// ---- VISUs/Modes/ProductionMode/V_ProductionBorgoFlaps.TcVIS
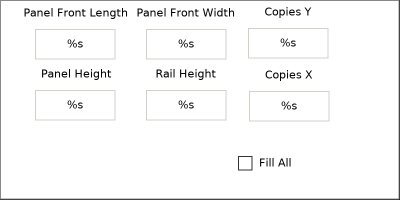
VISUALIZATION V_ProductionBorgoFlaps  // 400x200
VAR_IN_OUT
	HMI : ST_PackMLBaseModule_HMI;
	HMI_GantryXYZ : ST_GantryXYZ_HMI;
	HMI_Recipe : ST_RecipeBuilder_HMI;
END_VAR
    RoundedRectangle (0,0 400x200)
    Textfield (35,29 80x30), "%s", text variable: HMI_Recipe.Config.PanelFrontLength
        OnMouseClick: write the text variable via VisuDialogs.Numpad, min HMI_Recipe.Limits.PanelFrontLength.MinVal, max HMI_Recipe.Limits.PanelFrontLength.MaxVal
    Label (18,3 116x20), "Panel Front Length"
    Textfield (146,29 80x30), "%s", text variable: HMI_Recipe.Config.PanelFrontWidth
        OnMouseClick: write the text variable via VisuDialogs.Numpad, min HMI_Recipe.Limits.PanelFrontWidth.MinVal, max HMI_Recipe.Limits.PanelFrontWidth.MaxVal
    Label (97,3 178x20), "Panel Front Width"
    Textfield (35,90 80x30), "%s", text variable: HMI_Recipe.Config.PanelHeight
        OnMouseClick: write the text variable via VisuDialogs.Numpad, min HMI_Recipe.Limits.PanelHeight.MinVal, max HMI_Recipe.Limits.PanelHeight.MaxVal
    Label (19,64 115x20), "Panel Height"
    Textfield (146,90 80x30), "%s", text variable: HMI_Recipe.Config.RailHeightCorrection
        OnMouseClick: write the text variable via VisuDialogs.Numpad, min HMI_Recipe.Limits.RailHeightCorrection.MinVal, max HMI_Recipe.Limits.RailHeightCorrection.MaxVal
    Label (135,64 102x20), "Rail Height"
    Checkbox (236,148 72x30), "Fill All", variable: HMI_Recipe.Config.FillAll
    Textfield (249,91 80x30), "%s", text variable: HMI_Recipe.Config.RequestedCopiesX, input disabled if: MAIN.Seedra.RecipeConfig_HMI.Config.FillAll
        OnMouseClick: write the text variable via VisuDialogs.Numpad, min 1, max MAIN.Seedra.RecipeConfig_HMI.Limits.RequestedCopiesX.MaxVal
    Label (238,65 102x20), "Copies X"
    Textfield (248,28 80x30), "%s", text variable: HMI_Recipe.Config.RequestedCopiesY, input disabled if: MAIN.Seedra.RecipeConfig_HMI.Config.FillAll
        OnMouseClick: write the text variable via VisuDialogs.Numpad, min 1, max MAIN.Seedra.RecipeConfig_HMI.Limits.RequestedCopiesY.MaxVal
    Label (237,2 102x20), "Copies Y"
END_VISUALIZATION

// ---- VISUs/Modes/ProductionMode/V_ProductionBorgoWings.TcVIS
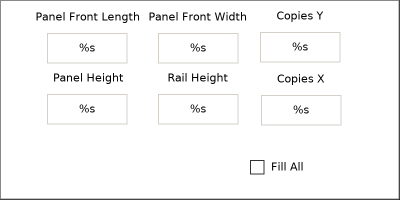
VISUALIZATION V_ProductionBorgoWings  // 400x200
VAR_IN_OUT
	HMI : ST_PackMLBaseModule_HMI;
	HMI_GantryXYZ : ST_GantryXYZ_HMI;
	HMI_Recipe : ST_RecipeBuilder_HMI;
END_VAR
    RoundedRectangle (0,0 400x200)
    Textfield (47,33 80x30), "%s", text variable: HMI_Recipe.Config.PanelFrontLength
        OnMouseClick: write the text variable via VisuDialogs.Numpad, min HMI_Recipe.Limits.PanelFrontLength.MinVal, max HMI_Recipe.Limits.PanelFrontLength.MaxVal
    Label (30,7 116x20), "Panel Front Length"
    Textfield (158,33 80x30), "%s", text variable: HMI_Recipe.Config.PanelFrontWidth
        OnMouseClick: write the text variable via VisuDialogs.Numpad, min HMI_Recipe.Limits.PanelFrontWidth.MinVal, max HMI_Recipe.Limits.PanelFrontWidth.MaxVal
    Label (109,7 178x20), "Panel Front Width"
    Textfield (47,94 80x30), "%s", text variable: HMI_Recipe.Config.PanelHeight
        OnMouseClick: write the text variable via VisuDialogs.Numpad, min HMI_Recipe.Limits.PanelHeight.MinVal, max HMI_Recipe.Limits.PanelHeight.MaxVal
    Label (31,68 115x20), "Panel Height"
    Textfield (158,94 80x30), "%s", text variable: HMI_Recipe.Config.RailHeightCorrection
        OnMouseClick: write the text variable via VisuDialogs.Numpad, min HMI_Recipe.Limits.RailHeightCorrection.MinVal, max HMI_Recipe.Limits.RailHeightCorrection.MaxVal
    Label (147,68 102x20), "Rail Height"
    Checkbox (248,152 72x30), "Fill All", variable: HMI_Recipe.Config.FillAll
    Textfield (261,95 80x30), "%s", text variable: HMI_Recipe.Config.RequestedCopiesX, input disabled if: MAIN.Seedra.RecipeConfig_HMI.Config.FillAll
        OnMouseClick: write the text variable via VisuDialogs.Numpad, min 1, max MAIN.Seedra.RecipeConfig_HMI.Limits.RequestedCopiesX.MaxVal
    Label (250,69 102x20), "Copies X"
    Textfield (260,32 80x30), "%s", text variable: HMI_Recipe.Config.RequestedCopiesY, input disabled if: MAIN.Seedra.RecipeConfig_HMI.Config.FillAll
        OnMouseClick: write the text variable via VisuDialogs.Numpad, min 1, max MAIN.Seedra.RecipeConfig_HMI.Limits.RequestedCopiesY.MaxVal
    Label (249,6 102x20), "Copies Y"
END_VISUALIZATION

// ---- VISUs/Modes/ProductionMode/V_Meina2_2000x1000.TcVIS
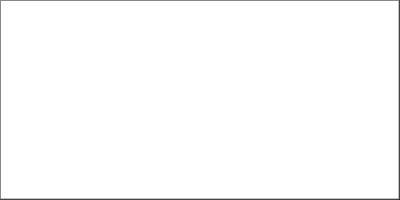
VISUALIZATION V_Meina2_2000x1000  // 400x200
VAR_IN_OUT
	HMI : ST_PackMLBaseModule_HMI;
	HMI_GantryXYZ : ST_GantryXYZ_HMI;
	HMI_Recipe : ST_RecipeBuilder_HMI;
END_VAR
    RoundedRectangle (0,0 400x200)
END_VISUALIZATION

// ---- VISUs/Modes/ProductionMode/V_ProductionWelcome.TcVIS
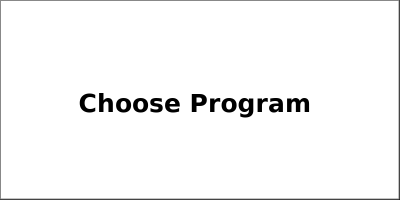
VISUALIZATION V_ProductionWelcome  // 400x200
    RoundedRectangle (0,0 400x200)
    Label (41,53 308x100), "Choose Program"
END_VISUALIZATION

// ---- VISUs/Modes/V_MaintenanceMode.TcVIS
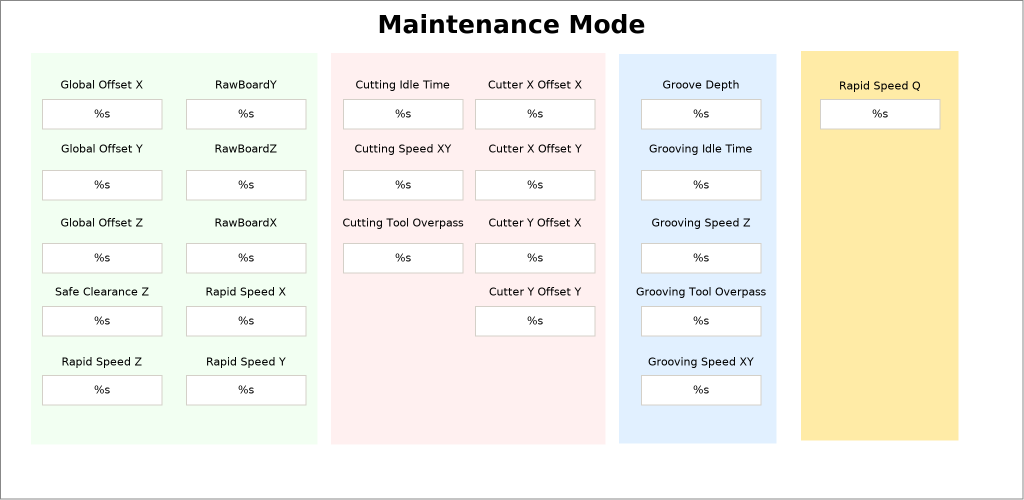
VISUALIZATION V_MaintenanceMode  // 1024x500
VAR_IN_OUT
	HMI : ST_PackMLBaseModule_HMI;
	HMI_GantryXYZ : ST_GantryXYZ_HMI;
	HMI_Recipe : ST_RecipeBuilder_HMI;
END_VAR
    Rectangle (30,52 288x393)
    Rectangle (330,52 276x393)
    Label (0,-1 1023x50), "Maintenance Mode"
    Rectangle (618,53 159x391)
    Textfield (641,99 120x30), "%s", text variable: HMI_Recipe.Config.GrooveDepthZ
        OnMouseClick: write the text variable via VisuDialogs.Numpad, min HMI_Recipe.Limits.GrooveDepthZ.MinVal, max HMI_Recipe.Limits.GrooveDepthZ.MaxVal
    Label (641,70 120x30), "Groove Depth"
    Textfield (641,306 120x30), "%s", text variable: HMI_Recipe.Config.GroovingOverpass
        OnMouseClick: write the text variable via VisuDialogs.Numpad, min HMI_Recipe.Limits.GroovingOverpass.MinVal, max HMI_Recipe.Limits.GroovingOverpass.MaxVal
    Label (641,277 120x30), "Grooving Tool Overpass"
    Textfield (641,375 120x30), "%s", text variable: HMI_GantryXYZ.Config.GroovingSpeedXY
        OnMouseClick: write the text variable via VisuDialogs.Numpad, min HMI_GantryXYZ.Limits.GroovingSpeedXY.MinVal, max HMI_GantryXYZ.Limits.GroovingSpeedXY.MaxVal
    Label (641,347 120x30), "Grooving Speed XY"
    Textfield (186,306 120x30), "%s", text variable: HMI_GantryXYZ.Config.RapidSpeedX
        OnMouseClick: write the text variable via VisuDialogs.Numpad, min HMI_GantryXYZ.Limits.RapidSpeedX.MinVal, max HMI_GantryXYZ.Limits.RapidSpeedX.MaxVal
    Label (186,277 120x30), "Rapid Speed X"
    Textfield (186,375 120x30), "%s", text variable: HMI_GantryXYZ.Config.RapidSpeedY
        OnMouseClick: write the text variable via VisuDialogs.Numpad, min HMI_GantryXYZ.Limits.RapidSpeedY.MinVal, max HMI_GantryXYZ.Limits.RapidSpeedY.MaxVal
    Label (186,347 120x30), "Rapid Speed Y"
    Textfield (641,243 120x30), "%s", text variable: HMI_GantryXYZ.Config.GroovingSpeedZ
        OnMouseClick: write the text variable via VisuDialogs.Numpad, min HMI_GantryXYZ.Limits.GroovingSpeedZ.MinVal, max HMI_GantryXYZ.Limits.GroovingSpeedZ.MaxVal
    Label (641,208 120x30), "Grooving Speed Z"
    Textfield (42,375 120x30), "%s", text variable: HMI_GantryXYZ.Config.RapidSpeedZ
        OnMouseClick: write the text variable via VisuDialogs.Numpad, min HMI_GantryXYZ.Limits.RapidSpeedZ.MinVal, max HMI_GantryXYZ.Limits.RapidSpeedZ.MaxVal
    Label (42,347 120x30), "Rapid Speed Z"
    Textfield (641,170 120x30), "%s", text variable: HMI_GantryXYZ.Config.GroovingIdleTime
        OnMouseClick: write the text variable via VisuDialogs.Numpad, min HMI_GantryXYZ.Limits.GroovingIdleTime.MinVal, max HMI_GantryXYZ.Limits.GroovingIdleTime.MaxVal
    Label (641,134 120x30), "Grooving Idle Time"
    Label (343,134 120x30), "Cutting Speed XY"
    Textfield (343,243 120x30), "%s", text variable: HMI_Recipe.Config.CuttingOverpass
        OnMouseClick: write the text variable via VisuDialogs.Numpad, min HMI_Recipe.Limits.CuttingOverpass.MinVal, max HMI_Recipe.Limits.CuttingOverpass.MaxVal
    Label (343,208 120x30), "Cutting Tool Overpass"
    Textfield (343,99 120x30), "%s", text variable: HMI_GantryXYZ.Config.CuttingIdleTime
        OnMouseClick: write the text variable via VisuDialogs.Numpad, min HMI_GantryXYZ.Limits.CuttingIdleTime.MinVal, max HMI_GantryXYZ.Limits.CuttingIdleTime.MaxVal
    Label (343,70 120x30), "Cutting Idle Time"
    Textfield (343,170 120x30), "%s", text variable: HMI_GantryXYZ.Config.CuttingSpeedXY
        OnMouseClick: write the text variable via VisuDialogs.Numpad, min HMI_GantryXYZ.Limits.CuttingSpeedXY.MinVal, max HMI_GantryXYZ.Limits.CuttingSpeedXY.MaxVal
    Label (475,70 120x30), "Cutter X Offset X"
    Textfield (475,170 120x30), "%s", text variable: HMI_GantryXYZ.Config.CutterXOffsetY
        OnMouseClick: write the text variable via VisuDialogs.Numpad, min HMI_GantryXYZ.Limits.CutterXOffsetY.MinVal, max HMI_GantryXYZ.Limits.CutterXOffsetY.MaxVal
    Label (475,134 120x30), "Cutter X Offset Y"
    Textfield (475,99 120x30), "%s", text variable: HMI_GantryXYZ.Config.CutterXOffsetX
        OnMouseClick: write the text variable via VisuDialogs.Numpad, min HMI_GantryXYZ.Limits.CutterXOffsetX.MinVal, max HMI_GantryXYZ.Limits.CutterXOffsetX.MaxVal
    Label (475,208 120x30), "Cutter Y Offset X"
    Textfield (475,306 120x30), "%s", text variable: HMI_GantryXYZ.Config.CutterYOffsetY
        OnMouseClick: write the text variable via VisuDialogs.Numpad, min HMI_GantryXYZ.Limits.CutterYOffsetY.MinVal, max HMI_GantryXYZ.Limits.CutterYOffsetY.MaxVal
    Label (475,277 120x30), "Cutter Y Offset Y"
    Textfield (475,243 120x30), "%s", text variable: HMI_GantryXYZ.Config.CutterYOffsetX
        OnMouseClick: write the text variable via VisuDialogs.Numpad, min HMI_GantryXYZ.Limits.CutterYOffsetX.MinVal, max HMI_GantryXYZ.Limits.CutterYOffsetX.MaxVal
    Label (42,70 120x30), "Global Offset X"
    Textfield (42,99 120x30), "%s", text variable: HMI_GantryXYZ.Config.GlobalOffsetX
        OnMouseClick: write the text variable via VisuDialogs.Numpad, min HMI_GantryXYZ.Limits.GlobalOffsetX.MinVal, max HMI_GantryXYZ.Limits.GlobalOffsetX.MaxVal
    Label (42,134 120x30), "Global Offset Y"
    Textfield (42,170 120x30), "%s", text variable: HMI_GantryXYZ.Config.GlobalOffsetY
        OnMouseClick: write the text variable via VisuDialogs.Numpad, min HMI_GantryXYZ.Limits.GlobalOffsetY.MinVal, max HMI_GantryXYZ.Limits.GlobalOffsetY.MaxVal
    Textfield (42,243 120x30), "%s", text variable: HMI_GantryXYZ.Config.GlobalOffsetZ
        OnMouseClick: write the text variable via VisuDialogs.Numpad, min HMI_GantryXYZ.Limits.GlobalOffsetZ.MinVal, max HMI_GantryXYZ.Limits.GlobalOffsetZ.MaxVal
    Label (42,208 120x30), "Global Offset Z"
    Textfield (186,243 120x30), "%s", text variable: HMI_GantryXYZ.Config.RawBoardX
        OnMouseClick: write the text variable via VisuDialogs.Numpad, min HMI_GantryXYZ.Limits.RawBoardX.MinVal, max HMI_GantryXYZ.Limits.RawBoardX.MaxVal
    Label (186,208 120x30), "RawBoardX"
    Textfield (186,99 120x30), "%s", text variable: HMI_GantryXYZ.Config.RawBoardY
        OnMouseClick: write the text variable via VisuDialogs.Numpad, min HMI_GantryXYZ.Limits.RawBoardY.MinVal, max HMI_GantryXYZ.Limits.RawBoardY.MaxVal
    Label (186,70 120x30), "RawBoardY"
    Textfield (186,170 120x30), "%s", text variable: HMI_GantryXYZ.Config.RawBoardZ
        OnMouseClick: write the text variable via VisuDialogs.Numpad, min HMI_GantryXYZ.Limits.RawBoardZ.MinVal, max HMI_GantryXYZ.Limits.RawBoardZ.MaxVal
    Label (186,134 120x30), "RawBoardZ"
    Textfield (42,306 120x30), "%s", text variable: HMI_GantryXYZ.Config.SafeClearanceZ
        OnMouseClick: write the text variable via VisuDialogs.Numpad, min HMI_GantryXYZ.Limits.SafeClearanceZ.MinVal, max HMI_GantryXYZ.Limits.SafeClearanceZ.MaxVal
    Label (42,277 120x30), "Safe Clearance Z"
    Rectangle (800,50 159x391)
    Textfield (820,99 120x30), "%s", text variable: HMI_GantryXYZ.Config.RapidSpeedQ
        OnMouseClick: write the text variable via VisuDialogs.Numpad, min HMI_GantryXYZ.Limits.RapidSpeedQ.MinVal, max HMI_GantryXYZ.Limits.RapidSpeedQ.MaxVal
    Label (820,71 120x30), "Rapid Speed Q"
END_VISUALIZATION

// ---- VISUs/Modes/V_ManualMode.TcVIS
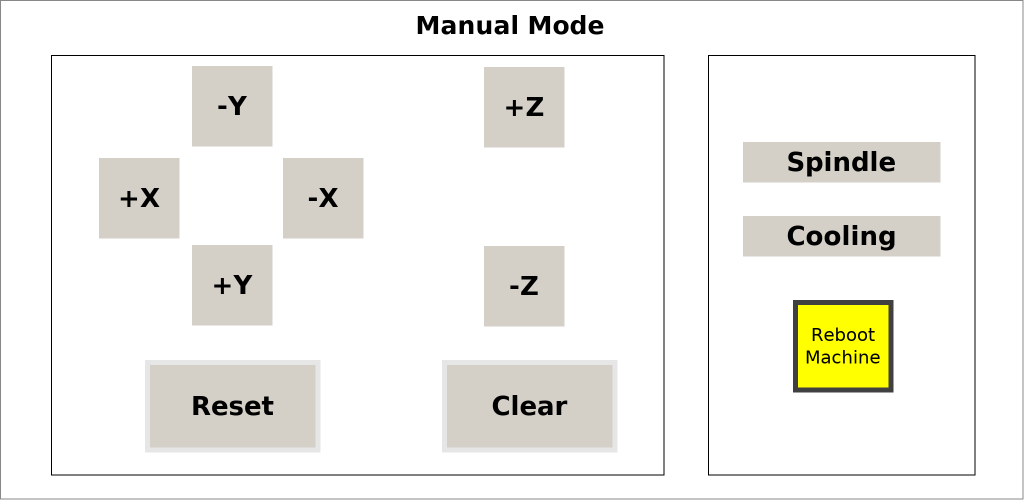
VISUALIZATION V_ManualMode  // 1024x500
VAR_IN_OUT
	HMI : ST_PackMLBaseModule_HMI;
	HMIAxeX : ST_AxisBase_HMI;
	HMIAxeY : ST_AxisBase_HMI;
	HMIAxeZ : ST_AxisBase_HMI;
END_VAR
    RoundedRectangle (51,55 613x420)
    RoundedRectangle (708,55 267x420)
    Label (0,0 1020x50), "Manual Mode"
    RoundedRectangle (738,137 207x50), "Spindle", colour toggle: HMI.Status.State = E_PMLState.ePMLState_Idle
        toggle SpindleEnable
    RoundedRectangle (738,211 207x50), "Cooling", colour toggle: HMI.Status.State = E_PMLState.ePMLState_Idle
        toggle CoolingEnable
    RoundedRectangle (283,158 80x80), "-X", colour toggle: HMI.Status.State = E_PMLState.ePMLState_Idle
        tap HMIAxeX.Command.JogFast_Backward
        OnMouseClick: execute { HMI.Command.State := E_PMLCommand.ePMLCommand_Clear; }
    RoundedRectangle (99,158 80x80), "+X", colour toggle: HMI.Status.State = E_PMLState.ePMLState_Idle
        tap HMIAxeX.Command.JogFast_Forward
    RoundedRectangle (192,245 80x80), "+Y", colour toggle: HMI.Status.State = E_PMLState.ePMLState_Idle
        tap HMIAxeY.Command.JogFast_Forward
    RoundedRectangle (192,66 80x80), "-Y", colour toggle: HMI.Status.State = E_PMLState.ePMLState_Idle
        tap HMIAxeY.Command.JogFast_Backward
        OnMouseClick: execute { HMI.Command.State := E_PMLCommand.ePMLCommand_Clear; }
    RoundedRectangle (484,67 80x80), "+Z", colour toggle: HMI.Status.State = E_PMLState.ePMLState_Idle
        tap HMIAxeZ.Command.JogSlow_Forward
    RoundedRectangle (484,246 80x80), "-Z", colour toggle: HMI.Status.State = E_PMLState.ePMLState_Idle
        tap HMIAxeZ.Command.JogSlow_Backward p3779583253=TRUE
    Rectangle (793,300 100x92), "Reboot Machine"
        OnMouseClick: execute { MAIN.RebootSystem(DELAY:=5,START:=TRUE); }
    RoundedRectangle (442,360 175x92), "Clear", colour toggle: (HMI.Status.State = E_PMLState.ePMLState_Aborted) OR (HMI.Status.State = E_PMLState.ePMLState_Clearing)
        OnMouseClick: execute { HMI.Command.State := E_PMLCommand.ePMLCommand_Clear; }
    RoundedRectangle (145,360 175x92), "Reset", colour toggle: (HMI.Status.State = E_PMLState.ePMLState_Complete) OR (HMI.Status.State = E_PMLState.ePMLState_Stopped) OR (HMI.Status.State = E_PMLState.ePMLState_Resetting)
        OnMouseClick: execute { HMI.Command.State := E_PMLCommand.ePMLCommand_Reset; }
END_VISUALIZATION

// ---- VISUs/Modes/V_ProductionMode.TcVIS
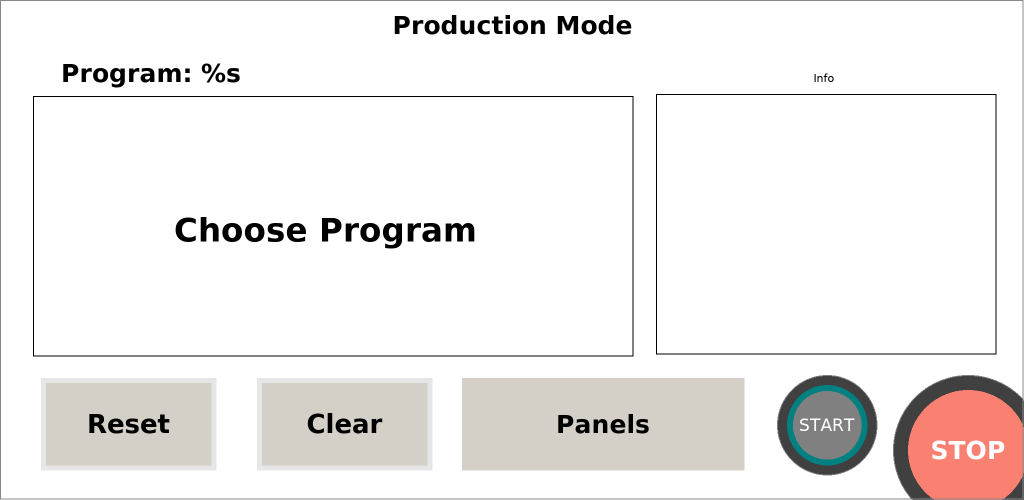
VISUALIZATION V_ProductionMode  // 1024x500
VAR_IN_OUT
	HMI : ST_PackMLBaseModule_HMI;
	HMI_GantryXYZ : ST_GantryXYZ_HMI;
	HMI_Recipe : ST_RecipeBuilder_HMI;
END_VAR
    Label (0,0 1025x50), "Production Mode"
    RoundedRectangle (257,378 175x92), "Clear", colour toggle: (HMI.Status.State = E_PMLState.ePMLState_Aborted) OR (HMI.Status.State = E_PMLState.ePMLState_Clearing)
        OnMouseClick: execute { HMI.Command.State := E_PMLCommand.ePMLCommand_Clear; }
    RoundedRectangle (41,378 175x92), "Reset", colour toggle: (HMI.Status.State = E_PMLState.ePMLState_Complete) OR (HMI.Status.State = E_PMLState.ePMLState_Stopped) OR (HMI.Status.State = E_PMLState.ePMLState_Resetting)
        OnMouseClick: execute { HMI.Command.State := E_PMLCommand.ePMLCommand_Reset; }
    Frame (33,96 600x260), frame switch variable: HMI_GantryXYZ.Command.ProgramIdRequested
        shows V_ProductionWelcome()
        shows V_ProductionBorgoFlaps(HMI := MAIN.Seedra.PackMLBaseModule_HMI, HMI_GantryXYZ := MAIN.Seedra.GantryXYZ.GantryXYZ_HMI, HMI_Recipe := MAIN.Seedra.RecipeConfig_HMI)
        shows V_ProductionBorgoWings(HMI := MAIN.Seedra.PackMLBaseModule_HMI, HMI_GantryXYZ := MAIN.Seedra.GantryXYZ.GantryXYZ_HMI, HMI_Recipe := MAIN.Seedra.RecipeConfig_HMI)
        shows V_ProductionArona(HMI := MAIN.Seedra.PackMLBaseModule_HMI, HMI_GantryXYZ := MAIN.Seedra.GantryXYZ.GantryXYZ_HMI, HMI_Recipe := MAIN.Seedra.RecipeConfig_HMI)
        shows V_ProductionNCICircle(HMI := MAIN.Seedra.PackMLBaseModule_HMI, HMI_GantryXYZ := MAIN.Seedra.GantryXYZ.GantryXYZ_HMI, HMI_Recipe := MAIN.Seedra.RecipeConfig_HMI)
        shows V_ProductionRectangle(HMI := MAIN.Seedra.PackMLBaseModule_HMI, HMI_GantryXYZ := MAIN.Seedra.GantryXYZ.GantryXYZ_HMI, HMI_Recipe := MAIN.Seedra.RecipeConfig_HMI)
        shows V_ProductionRoundRectangle(HMI := MAIN.Seedra.PackMLBaseModule_HMI, HMI_GantryXYZ := MAIN.Seedra.GantryXYZ.GantryXYZ_HMI, HMI_Recipe := MAIN.Seedra.RecipeConfig_HMI)
        shows V_ProductionFeedCircle(HMI := MAIN.Seedra.PackMLBaseModule_HMI, HMI_GantryXYZ := MAIN.Seedra.GantryXYZ.GantryXYZ_HMI, HMI_Recipe := MAIN.Seedra.RecipeConfig_HMI)
        shows V_Meina2_2000x1000(HMI := MAIN.Seedra.PackMLBaseModule_HMI, HMI_GantryXYZ := MAIN.Seedra.GantryXYZ.GantryXYZ_HMI, HMI_Recipe := MAIN.Seedra.RecipeConfig_HMI)
        shows V_ProductionMeina2_5Squares(HMI := MAIN.Seedra.PackMLBaseModule_HMI, HMI_GantryXYZ := MAIN.Seedra.GantryXYZ.GantryXYZ_HMI, HMI_Recipe := MAIN.Seedra.RecipeConfig_HMI)
        shows V_ProductionMeina2_5Circles(HMI := MAIN.Seedra.PackMLBaseModule_HMI, HMI_GantryXYZ := MAIN.Seedra.GantryXYZ.GantryXYZ_HMI, HMI_Recipe := MAIN.Seedra.RecipeConfig_HMI)
        shows V_ProductionMeina2_3Squares(HMI := MAIN.Seedra.PackMLBaseModule_HMI, HMI_GantryXYZ := MAIN.Seedra.GantryXYZ.GantryXYZ_HMI, HMI_Recipe := MAIN.Seedra.RecipeConfig_HMI)
        shows V_ProductionMeina2_3Circles(HMI := MAIN.Seedra.PackMLBaseModule_HMI, HMI_GantryXYZ := MAIN.Seedra.GantryXYZ.GantryXYZ_HMI, HMI_Recipe := MAIN.Seedra.RecipeConfig_HMI)
        shows V_ProductionMeina2_2Squares(HMI := MAIN.Seedra.PackMLBaseModule_HMI, HMI_GantryXYZ := MAIN.Seedra.GantryXYZ.GantryXYZ_HMI, HMI_Recipe := MAIN.Seedra.RecipeConfig_HMI)
        shows V_ProductionMeina2_2Circles(HMI := MAIN.Seedra.PackMLBaseModule_HMI, HMI_GantryXYZ := MAIN.Seedra.GantryXYZ.GantryXYZ_HMI, HMI_Recipe := MAIN.Seedra.RecipeConfig_HMI)
        shows V_ProductionMeina2_2Rectangles(HMI := MAIN.Seedra.PackMLBaseModule_HMI, HMI_GantryXYZ := MAIN.Seedra.GantryXYZ.GantryXYZ_HMI, HMI_Recipe := MAIN.Seedra.RecipeConfig_HMI)
        shows V_Meina2_Samples(HMI := MAIN.Seedra.PackMLBaseModule_HMI, HMI_GantryXYZ := MAIN.Seedra.GantryXYZ.GantryXYZ_HMI, HMI_Recipe := MAIN.Seedra.RecipeConfig_HMI)
        p3843536458: MAIN.Seedra.RecipeBuilderWings.RecipeBuilder_HMI
    RoundedRectangle (656,94 340x260)
    Group (893,375 100x100)
        Ellipse (0,0 150x150)
        Ellipse (15,15 120x120), "STOP"
            toggle GVL_Safety.eStopHMI
    Label (679,66 290x25), "Info"
    RoundedRectangle (462,378 282x92), "Panels"
        OnMouseClick: execute { GVL_HMI.PopupToDisplay := 2; }
    Textfield (58,57 531x32), "Program: %s", text variable: MAIN.Seedra.sSelectedRecipeName
    Ellipse (777,375 100x100)
    Ellipse (787,385 80x80), "START", colour toggle: HMI.Status.State = E_PMLState.ePMLState_Idle, input disabled if: NOT MAIN.Seedra.RecipeConfig_HMI.Config.IsValid
        OnMouseClick: execute { HMI.Command.State := E_PMLCommand.ePMLCommand_Start; }
END_VISUALIZATION

// ---- VISUs/V_InfoMenu.TcVIS
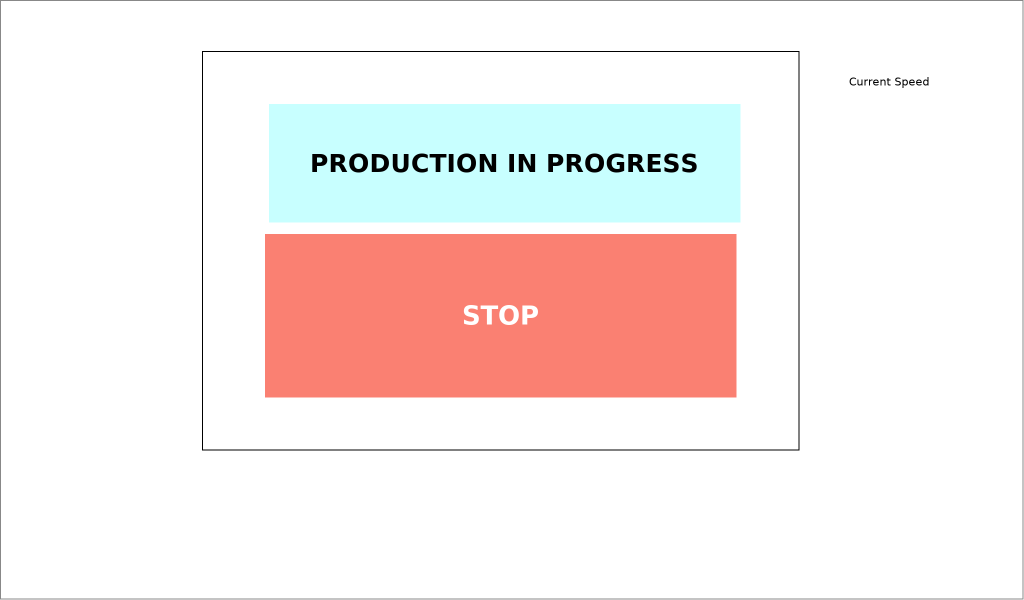
VISUALIZATION V_InfoMenu  // 1024x600
    RoundedRectangle (202,51 597x399)
    RoundedRectangle (268,103 473x120), "PRODUCTION IN PROGRESS"
    RoundedRectangle (264,233 473x165), "STOP"
        toggle GVL_Safety.eStopHMI
    Label (829,67 121x30), "Current Speed"
END_VISUALIZATION

// ---- VISUs/V_MainMenu.TcVIS
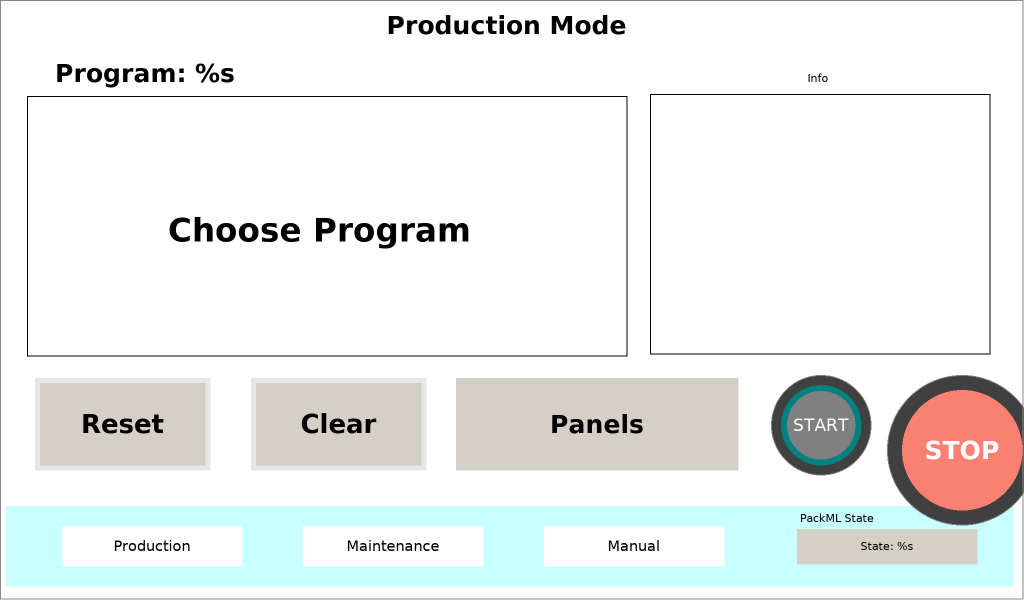
VISUALIZATION V_MainMenu  // 1024x600
VAR_IN_OUT
	HMI : ST_PackMLBaseModule_HMI;
	HMIAxeX : ST_AxisBase_HMI;
	HMI_Recipe : ST_RecipeBuilder_HMI;
	HMI2 : ST_Machine_HMI;
END_VAR
    RoundedRectangle (5,505 1009x82)
    Textfield (797,529 180x35), "State: %s", text variable: HMI2.Status.PackMLState
    RoundedRectangle (62,526 180x40), "Production", colour toggle: HMI.Status.Mode = E_PMLUnitMode.ePMLUnitMode_Production
        OnMouseClick: execute { HMI.Command.Mode := E_PMLUnitMode.ePMLUnitMode_Production; }
    RoundedRectangle (303,526 180x40), "Maintenance", colour toggle: HMI.Status.Mode = E_PMLUnitMode.ePMLUnitMode_Maintenance
        OnMouseClick: execute { HMI.Command.Mode := E_PMLUnitMode.ePMLUnitMode_Maintenance; }
    RoundedRectangle (544,526 180x40), "Manual", colour toggle: HMI.Status.Mode = E_PMLUnitMode.ePMLUnitMode_Manual
        OnMouseClick: execute { HMI.Command.Mode := E_PMLUnitMode.ePMLUnitMode_Manual; }
    Frame (-6,0 1024x500), frame switch variable: GVL_HMI.MenuToDisplay
        shows V_ProductionMode(HMI := MAIN.Seedra.PackMLBaseModule_HMI, HMI_GantryXYZ := MAIN.Seedra.GantryXYZ.GantryXYZ_HMI, HMI_Recipe := MAIN.Seedra.RecipeConfig_HMI)
        shows V_ManualMode(HMI := MAIN.Seedra.PackMLBaseModule_HMI, HMIAxeX := MAIN.Seedra.GantryXYZ.AxisX.AxisBase_HMI, HMIAxeY := MAIN.Seedra.GantryXYZ.AxisY.AxisBase_HMI, HMIAxeZ := MAIN.Seedra.GantryXYZ.AxisZ.AxisBase_HMI)
        shows V_MaintenanceMode(HMI := MAIN.Seedra.PackMLBaseModule_HMI, HMI_GantryXYZ := MAIN.Seedra.GantryXYZ.GantryXYZ_HMI, HMI_Recipe := MAIN.Seedra.RecipeConfig_HMI)
    Label (788,498 98x41), "PackML State"
END_VISUALIZATION

// ---- VISUs/V_Main.TcVIS
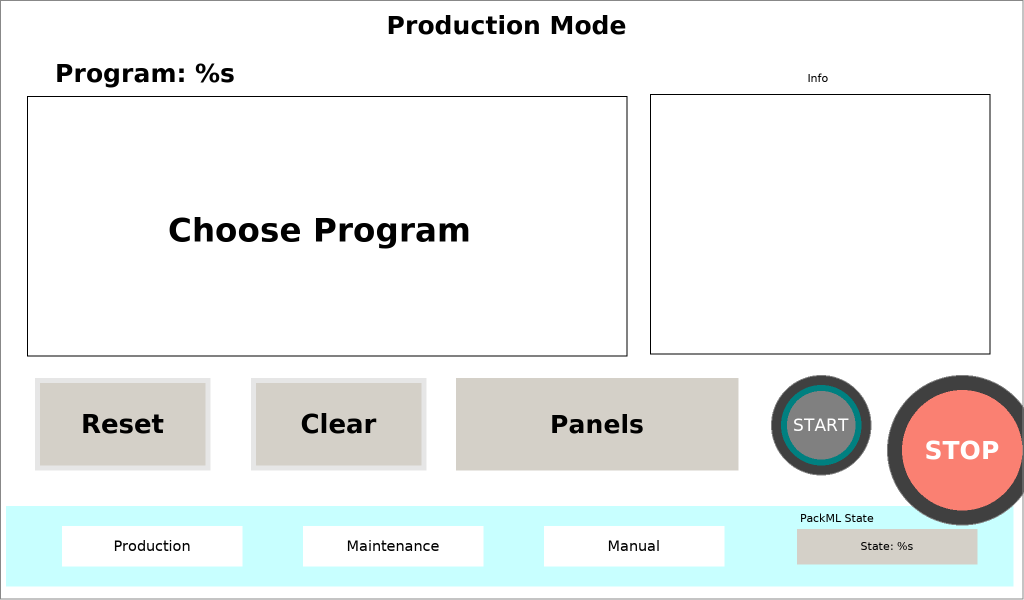
VISUALIZATION V_Main  // 1024x600
    Frame (0,0 1024x600), frame switch variable: GVL_HMI.PopupToDisplay
        shows V_MainMenu(HMI := MAIN.Seedra.PackMLBaseModule_HMI, HMIAxeX := MAIN.Seedra.GantryXYZ.AxisX.AxisBase_HMI, HMI_Recipe := MAIN.Seedra.RecipeConfig_HMI, HMI2 := MAIN.Seedra.Machine_HMI)
        shows V_InfoMenu()
        shows V_Builders(HMI := MAIN.Seedra.PackMLBaseModule_HMI, HMI_GantryXYZ := MAIN.Seedra.GantryXYZ.GantryXYZ_HMI)
END_VISUALIZATION
